FUNCTION_BLOCK FB_ROR_BYTE
  (* Standard: 61131-3 *)
  (* Version 0.1, 2007-04-02, JHC, Holobloc Inc, Added missing REQ/CNF interface, corrected package. *)
  (* Version 0.0, 2004-12-15, JHC, Rockwell Automation, Converted from SRC format. *)
  (* Compiler header: package fb.rt.math; *)
  (* Compiler Java Sun JDK 1.6.0 *)
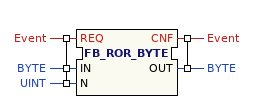
  EVENT_INPUT
    REQ WITH IN, N;
  END_EVENT
  EVENT_OUTPUT
    CNF WITH OUT;
  END_EVENT
  VAR_INPUT
    IN : BYTE;
    N : UINT;
  END_VAR
  VAR_OUTPUT
    OUT : BYTE;
  END_VAR
END_FUNCTION_BLOCK
